ABB RAPID module: HardcodedTargets.mod

MODULE HardcodedTargets

    CONST robtarget Home:=[[1000.00, 0.00, 1000.00 ],[0,0,1,0],[0,0,0,0],[9E+09,9E+09,9E+09,9E+09,9E+09,9E+09]];

    CONST robtarget Pick_0:=[[1030.00, -734.50, 980.00 ],[0,0,1,0],[0,0,0,0],[9E+09,9E+09,9E+09,9E+09,9E+09,9E+09]];
    CONST robtarget Pick_2:=[[758.07, -734.39, 829.70 ],[0,0,1,0],[0,0,0,0],[9E+09,9E+09,9E+09,9E+09,9E+09,9E+09]];
    CONST robtarget Pick_1:=[[1031.58, -734.39, 829.70 ],[0,0,1,0],[0,0,0,0],[9E+09,9E+09,9E+09,9E+09,9E+09,9E+09]];
    CONST robtarget Pick_3:=[[1301.80, -734.39, 829.70 ],[0,0,1,0],[0,0,0,0],[9E+09,9E+09,9E+09,9E+09,9E+09,9E+09]];
    CONST robtarget Pick_5:=[[756.82, -734.87, 376.55 ],[0,0,1,0],[0,0,0,0],[9E+09,9E+09,9E+09,9E+09,9E+09,9E+09]];
    CONST robtarget Pick_4:=[[1034.75, -734.87, 376.55 ],[0,0,1,0],[0,0,0,0],[9E+09,9E+09,9E+09,9E+09,9E+09,9E+09]];
    CONST robtarget Pick_6:=[[1304.10, -734.87, 376.55 ],[0,0,1,0],[0,0,0,0],[9E+09,9E+09,9E+09,9E+09,9E+09,9E+09]];
    CONST robtarget Pick_8:=[[756.62, -734.87, 435.05 ],[0,0,1,0],[0,0,0,0],[9E+09,9E+09,9E+09,9E+09,9E+09,9E+09]];
    CONST robtarget Pick_7:=[[1034.96, -734.87, 435.05 ],[0,0,1,0],[0,0,0,0],[9E+09,9E+09,9E+09,9E+09,9E+09,9E+09]];
    CONST robtarget Pick_9:=[[1311.78, -734.87, 435.05 ],[0,0,1,0],[0,0,0,0],[9E+09,9E+09,9E+09,9E+09,9E+09,9E+09]];
    CONST robtarget Pick_11:=[[755.98, -734.67, 490.10 ],[0,0,1,0],[0,0,0,0],[9E+09,9E+09,9E+09,9E+09,9E+09,9E+09]];
    CONST robtarget Pick_10:=[[1034.44, -734.67, 490.10 ],[0,0,1,0],[0,0,0,0],[9E+09,9E+09,9E+09,9E+09,9E+09,9E+09]];
    CONST robtarget Pick_12:=[[1306.63, -734.67, 490.10 ],[0,0,1,0],[0,0,0,0],[9E+09,9E+09,9E+09,9E+09,9E+09,9E+09]];
    CONST robtarget Pick_14:=[[755.93, -734.87, 544.35 ],[0,0,1,0],[0,0,0,0],[9E+09,9E+09,9E+09,9E+09,9E+09,9E+09]];
    CONST robtarget Pick_13:=[[1032.55, -734.87, 544.35 ],[0,0,1,0],[0,0,0,0],[9E+09,9E+09,9E+09,9E+09,9E+09,9E+09]];
    CONST robtarget Pick_15:=[[1306.44, -734.87, 544.35 ],[0,0,1,0],[0,0,0,0],[9E+09,9E+09,9E+09,9E+09,9E+09,9E+09]];
    CONST robtarget Pick_17:=[[757.79, -735.97, 600.81 ],[0,0,1,0],[0,0,0,0],[9E+09,9E+09,9E+09,9E+09,9E+09,9E+09]];
    CONST robtarget Pick_16:=[[1035.85, -735.97, 600.81 ],[0,0,1,0],[0,0,0,0],[9E+09,9E+09,9E+09,9E+09,9E+09,9E+09]];
    CONST robtarget Pick_18:=[[1306.18, -735.97, 600.81 ],[0,0,1,0],[0,0,0,0],[9E+09,9E+09,9E+09,9E+09,9E+09,9E+09]];
    CONST robtarget Pick_20:=[[756.28, -734.57, 661.68 ],[0,0,1,0],[0,0,0,0],[9E+09,9E+09,9E+09,9E+09,9E+09,9E+09]];
    CONST robtarget Pick_19:=[[1028.66, -734.57, 661.68 ],[0,0,1,0],[0,0,0,0],[9E+09,9E+09,9E+09,9E+09,9E+09,9E+09]];
    CONST robtarget Pick_21:=[[1303.40, -734.57, 661.68 ],[0,0,1,0],[0,0,0,0],[9E+09,9E+09,9E+09,9E+09,9E+09,9E+09]];
    CONST robtarget Pick_23:=[[756.08, -734.44, 715.52 ],[0,0,1,0],[0,0,0,0],[9E+09,9E+09,9E+09,9E+09,9E+09,9E+09]];
    CONST robtarget Pick_22:=[[1026.11, -734.44, 715.52 ],[0,0,1,0],[0,0,0,0],[9E+09,9E+09,9E+09,9E+09,9E+09,9E+09]];
    CONST robtarget Pick_24:=[[1300.55, -734.44, 715.52 ],[0,0,1,0],[0,0,0,0],[9E+09,9E+09,9E+09,9E+09,9E+09,9E+09]];
    CONST robtarget Pick_26:=[[759.70, -734.41, 772.95 ],[0,0,1,0],[0,0,0,0],[9E+09,9E+09,9E+09,9E+09,9E+09,9E+09]];
    CONST robtarget Pick_25:=[[1025.89, -734.41, 772.95 ],[0,0,1,0],[0,0,0,0],[9E+09,9E+09,9E+09,9E+09,9E+09,9E+09]];
    CONST robtarget Pick_27:=[[1304.37, -734.41, 772.95 ],[0,0,1,0],[0,0,0,0],[9E+09,9E+09,9E+09,9E+09,9E+09,9E+09]];

    CONST robtarget Place_0:=[[1050.00,500.00,760.00],[0.0000,0.2696,0.9630,0.0000],[0,0,0,0],[9E+09,9E+09,9E+09,9E+09,9E+09,9E+09]];
    CONST robtarget Place_1:=[[595.24,727.44,390.00],[0.0000,0.2696,0.9630,0.0000],[0,0,0,0],[9E+09,9E+09,9E+09,9E+09,9E+09,9E+09]];
    CONST robtarget Place_2:=[[825.98,587.24,390.00],[0.0000,0.3952,0.9186,0.0000],[0,0,0,0],[9E+09,9E+09,9E+09,9E+09,9E+09,9E+09]];
    CONST robtarget Place_3:=[[1056.73,447.03,390.00],[0.0000,0.6213,0.7836,0.0000],[0,0,0,0],[9E+09,9E+09,9E+09,9E+09,9E+09,9E+09]];
    CONST robtarget Place_4:=[[1287.47,306.83,390.00],[0.0000,0.3952,0.9186,0.0000],[0,0,0,0],[9E+09,9E+09,9E+09,9E+09,9E+09,9E+09]];
    CONST robtarget Place_5:=[[1518.22,166.63,390.00],[0.0000,0.2696,0.9630,0.0000],[0,0,0,0],[9E+09,9E+09,9E+09,9E+09,9E+09,9E+09]];
    CONST robtarget Place_6:=[[710.61,657.34,445.00],[0.0000,0.3952,0.9186,0.0000],[0,0,0,0],[9E+09,9E+09,9E+09,9E+09,9E+09,9E+09]];
    CONST robtarget Place_7:=[[941.36,517.13,445.00],[0.0000,0.6213,0.7836,0.0000],[0,0,0,0],[9E+09,9E+09,9E+09,9E+09,9E+09,9E+09]];
    CONST robtarget Place_8:=[[1172.10,376.93,445.00],[0.0000,0.3952,0.9186,0.0000],[0,0,0,0],[9E+09,9E+09,9E+09,9E+09,9E+09,9E+09]];
    CONST robtarget Place_9:=[[1402.85,236.73,445.00],[0.0000,0.2696,0.9630,0.0000],[0,0,0,0],[9E+09,9E+09,9E+09,9E+09,9E+09,9E+09]];
    CONST robtarget Place_10:=[[1569.23,135.63,445.00],[0.0000,-0.4903,0.8716,0.0000],[0,0,0,0],[9E+09,9E+09,9E+09,9E+09,9E+09,9E+09]];
    CONST robtarget Place_11:=[[544.23,758.44,445.00],[0.0000,-0.4903,0.8716,0.0000],[0,0,0,0],[9E+09,9E+09,9E+09,9E+09,9E+09,9E+09]];
    CONST robtarget Place_12:=[[595.24,727.44,500.00],[0.0000,0.2696,0.9630,0.0000],[0,0,0,0],[9E+09,9E+09,9E+09,9E+09,9E+09,9E+09]];
    CONST robtarget Place_13:=[[825.98,587.24,500.00],[0.0000,0.3952,0.9186,0.0000],[0,0,0,0],[9E+09,9E+09,9E+09,9E+09,9E+09,9E+09]];
    CONST robtarget Place_14:=[[1056.73,447.03,500.00],[0.0000,0.6213,0.7836,0.0000],[0,0,0,0],[9E+09,9E+09,9E+09,9E+09,9E+09,9E+09]];
    CONST robtarget Place_15:=[[1287.47,306.83,500.00],[0.0000,0.5132,0.8583,0.0000],[0,0,0,0],[9E+09,9E+09,9E+09,9E+09,9E+09,9E+09]];
    CONST robtarget Place_16:=[[1518.22,166.63,500.00],[0.0000,0.2696,0.9630,0.0000],[0,0,0,0],[9E+09,9E+09,9E+09,9E+09,9E+09,9E+09]];
    CONST robtarget Place_17:=[[710.61,657.34,555.00],[0.0000,0.3952,0.9186,0.0000],[0,0,0,0],[9E+09,9E+09,9E+09,9E+09,9E+09,9E+09]];
    CONST robtarget Place_18:=[[941.36,517.13,555.00],[0.0000,0.6213,0.7836,0.0000],[0,0,0,0],[9E+09,9E+09,9E+09,9E+09,9E+09,9E+09]];
    CONST robtarget Place_19:=[[1172.10,376.93,555.00],[0.0000,0.5132,0.8583,0.0000],[0,0,0,0],[9E+09,9E+09,9E+09,9E+09,9E+09,9E+09]];
    CONST robtarget Place_20:=[[1402.85,236.73,555.00],[0.0000,0.2696,0.9630,0.0000],[0,0,0,0],[9E+09,9E+09,9E+09,9E+09,9E+09,9E+09]];
    CONST robtarget Place_21:=[[1569.23,135.63,555.00],[0.0000,-0.4903,0.8716,0.0000],[0,0,0,0],[9E+09,9E+09,9E+09,9E+09,9E+09,9E+09]];
    CONST robtarget Place_22:=[[544.23,758.44,555.00],[0.0000,-0.4903,0.8716,0.0000],[0,0,0,0],[9E+09,9E+09,9E+09,9E+09,9E+09,9E+09]];
    CONST robtarget Place_23:=[[595.24,727.44,610.00],[0.0000,0.2696,0.9630,0.0000],[0,0,0,0],[9E+09,9E+09,9E+09,9E+09,9E+09,9E+09]];
    CONST robtarget Place_24:=[[825.98,587.24,610.00],[0.0000,0.2696,0.9630,0.0000],[0,0,0,0],[9E+09,9E+09,9E+09,9E+09,9E+09,9E+09]];
    CONST robtarget Place_25:=[[1056.73,447.03,610.00],[0.0000,0.6213,0.7836,0.0000],[0,0,0,0],[9E+09,9E+09,9E+09,9E+09,9E+09,9E+09]];
    CONST robtarget Place_26:=[[1287.47,306.83,610.00],[0.0000,0.5132,0.8583,0.0000],[0,0,0,0],[9E+09,9E+09,9E+09,9E+09,9E+09,9E+09]];
    CONST robtarget Place_27:=[[1518.22,166.63,610.00],[0.0000,0.2696,0.9630,0.0000],[0,0,0,0],[9E+09,9E+09,9E+09,9E+09,9E+09,9E+09]];

ENDMODULE
